Fanuc KAREL source: compact_preamble.KL

PROGRAM IO0039
%NOLOCKGROUP
ROUTINE RTEST
VAR
L1 : ARRAY[3] OF INTEGER;L2 : XYZWPR
L3 : JOINTPOS9
L4 : POSITION
S1:INTEGER
A:REAL
B:REAL
C:BOOLEAN
D:REAL
BEGIN
S1=1
L1[1]=2
C=TRUE
D=1.0
IF (GIN[17] > 0) THEN
S1=(S1 + 1)
ENDIF
END RTEST
BEGIN
RTEST
END IO0039
